(* PLC project Sin nombre, Desconocido Sin nombre 1 *)
(* stored: creationDateTime 2020-09-15T17:35:25, modificationDateTime 2025-01-28T11:14:47 *)

PROGRAM program0
  VAR
    B1_AL : BOOL;
    B1_AB : BOOL;
    B1_CE : BOOL;
    B1_ST_SALA : BOOL;
    B1_ST_POZO : BOOL;
    B1_Q : BOOL;
    B2_AL : BOOL;
    B2_AB : BOOL;
    B2_CE : BOOL;
    B2_ST_SALA : BOOL;
    B2_ST_POZO : BOOL;
    B2_Q : BOOL;
    SEL_SALA : BOOL;
    CDO_AR_SALA : BOOL;
    CDO_PAR_SALA : BOOL;
    FALLA_SALA : BOOL;
    SEL_POZO : BOOL;
    CDO_AR_POZO : BOOL;
    CDO_PAR_POZO : BOOL;
    FALLA_POZO : BOOL;
    CAUDAL : REAL;
    AUX_ARRANQUE : BOOL;
  END_VAR

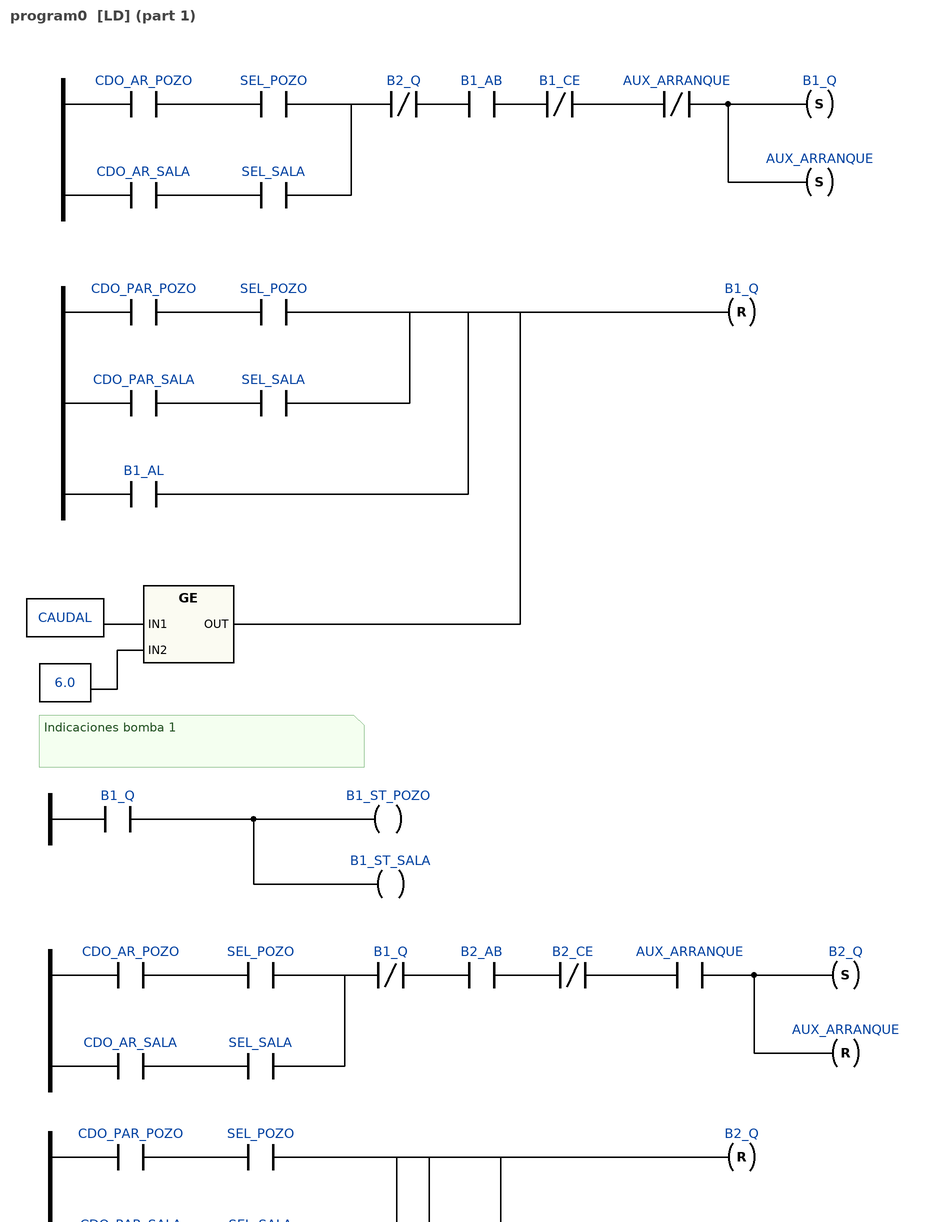
(* LD diagram, written out as Structured Text *)
IF (CDO_AR_POZO AND SEL_POZO OR CDO_AR_SALA AND SEL_SALA) AND NOT B2_Q AND B1_AB AND NOT B1_CE AND NOT AUX_ARRANQUE THEN B1_Q := TRUE; END_IF;
IF CDO_PAR_POZO AND SEL_POZO OR CDO_PAR_SALA AND SEL_SALA OR B1_AL OR CAUDAL >= 6.0 THEN B1_Q := FALSE; END_IF;
(* Indicaciones bomba 1 *)
IF CDO_PAR_POZO AND SEL_POZO OR CDO_PAR_SALA AND SEL_SALA OR B2_AL OR CAUDAL >= 6.0 THEN B2_Q := FALSE; END_IF;
IF (CDO_AR_POZO AND SEL_POZO OR CDO_AR_SALA AND SEL_SALA) AND NOT B1_Q AND B2_AB AND NOT B2_CE AND AUX_ARRANQUE THEN B2_Q := TRUE; END_IF;
IF (CDO_AR_POZO AND SEL_POZO OR CDO_AR_SALA AND SEL_SALA) AND NOT B2_Q AND B1_AB AND NOT B1_CE AND NOT AUX_ARRANQUE THEN AUX_ARRANQUE := TRUE; END_IF;
IF (CDO_AR_POZO AND SEL_POZO OR CDO_AR_SALA AND SEL_SALA) AND NOT B1_Q AND B2_AB AND NOT B2_CE AND AUX_ARRANQUE THEN AUX_ARRANQUE := FALSE; END_IF;
B1_ST_POZO := B1_Q;
B1_ST_SALA := B1_Q;
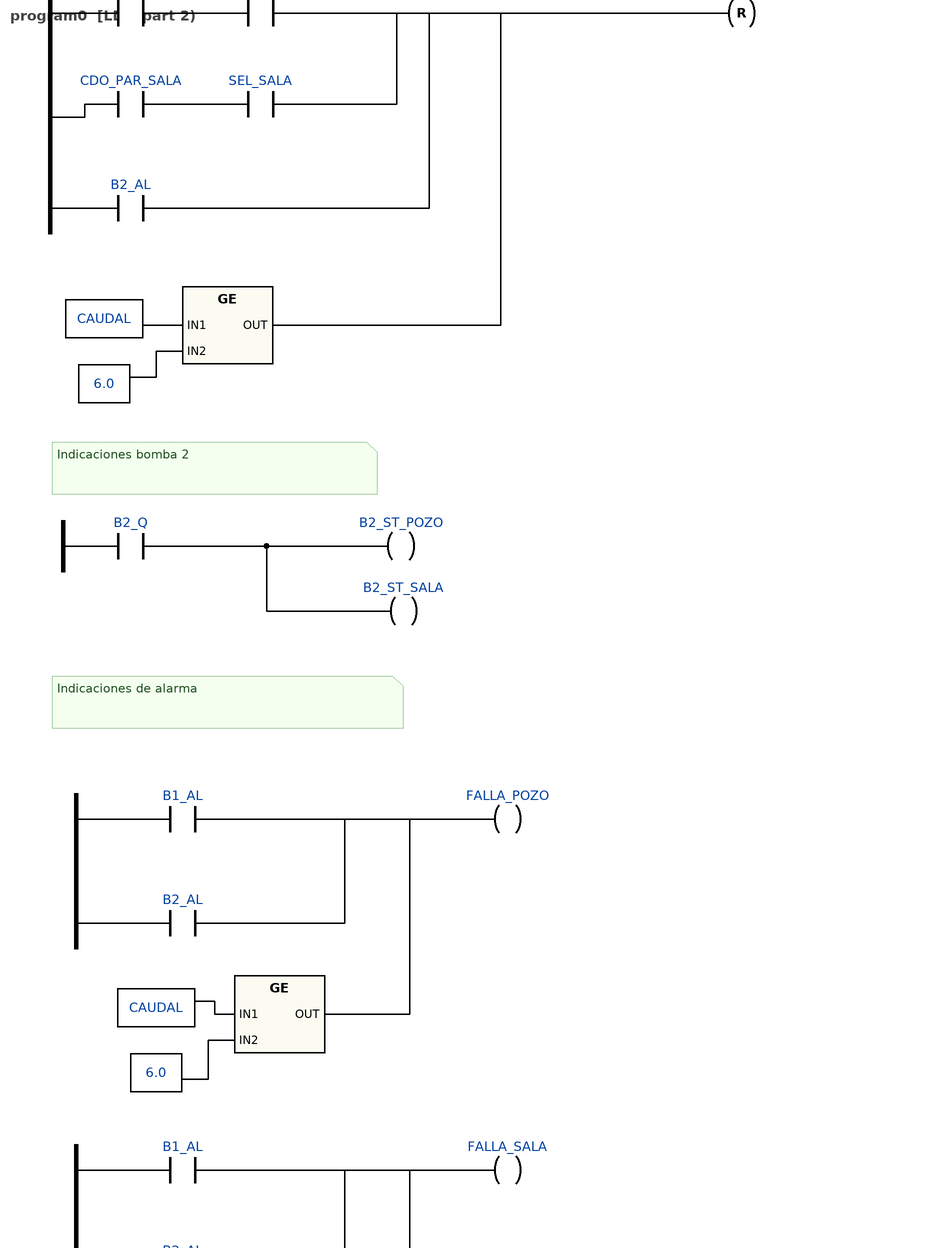
(* Indicaciones bomba 2 *)
B2_ST_POZO := B2_Q;
B2_ST_SALA := B2_Q;
(* Indicaciones de alarma *)
FALLA_POZO := B1_AL OR B2_AL OR CAUDAL >= 6.0;
FALLA_SALA := B1_AL OR B2_AL OR CAUDAL >= 6.0;
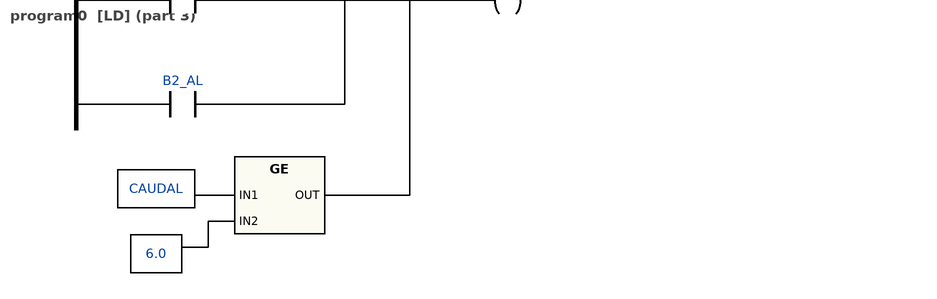
END_PROGRAM

CONFIGURATION Config0
  RESOURCE Res0 ON PLC
    TASK task0(INTERVAL := T#20ms, PRIORITY := 0);
    PROGRAM instance0 WITH task0 : program0;
  END_RESOURCE
END_CONFIGURATION
